FUNCTION_BLOCK Fan
VAR_INPUT
END_VAR
VAR_OUTPUT
END_VAR
VAR
END_VAR

END_FUNCTION_BLOCK

(* stored: Version 1.1.0.1, ProductVersion 3.1.4024.13
   POU Fan: Id {83141499-b7a6-42a6-9529-a95faf7cf666}, SpecialFunc None *)
